{attribute clr[Container(Layout.Stack)]}
{attribute clr[Group(Layout.GroupBox)]}
{attribute addProperty PreviousPort "Unknown"}
TYPE EtcSlaveTerminalBase_947E5A46 :
STRUCT
END_STRUCT
END_TYPE

(* stored: Version 1.2.0.0, ProductVersion 3.1.4024.9
   DUT EtcSlaveTerminalBase_947E5A46: Id {b0b78b44-a08f-4d16-a645-8f802923a2bf} *)
